FUNCTION_BLOCK EA_network1
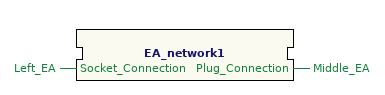
  SOCKETS
    Socket_Connection : Left_EA;
  END_SOCKETS
  PLUGS
    Plug_Connection : Middle_EA;
  END_PLUGS
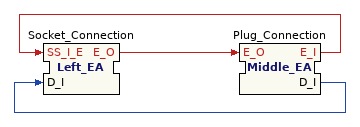
  EVENT_CONNECTIONS
    Socket_Connection.E_O TO Plug_Connection.E_O;
    Plug_Connection.E_I TO Socket_Connection.SS_I_E;
  END_CONNECTIONS
  DATA_CONNECTIONS
    Plug_Connection.D_I TO Socket_Connection.D_I;
  END_CONNECTIONS
END_FUNCTION_BLOCK
